{attribute 'pack_mode' := '2'}
TYPE ST_XPU_CTRL :
STRUCT
  Cmd             : E_XPU_CTRL;
END_STRUCT
END_TYPE

(* stored: Version 1.1.0.1
   DUT ST_XPU_CTRL: Id {3a097616-64f3-425e-a1f4-8c0dec770ddb} *)
